// Mitsubishi GX Works2 project: z14   PLC: Q02/Q02H

PROGRAM MAIN
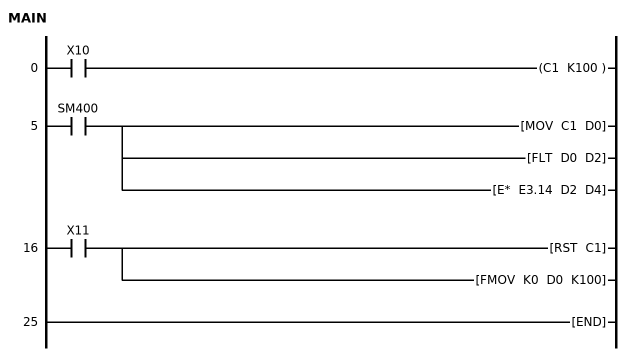
0     LD      X10
      OUT     C1 K100
5     LD      SM400
      MOV     C1 D0
      FLT     D0 D2
      E*      E3.14 D2 D4
16    LD      X11
      RST     C1
      FMOV    K0 D0 K100
25    END
END_PROGRAM
